// TIA Portal V19 export
TYPE "PQI_IF"
   STRUCT
      O_DI4 : Bool;   // Output signal status Pin 4
      O_DI2 : Bool;   // Output signal status Pin 2
      O_DA : Bool;   // Output device recognized
      O_DE : Bool;   // Output device error event has appeared
      O_PQ : Bool;   // Output port qualifer process data valid
   END_STRUCT;
END_TYPE
